TYPE ERROR :
STRUCT
	bError : BOOL;
	nErrorCode : UDINT;
	dtCurrentTime : DT;
END_STRUCT
END_TYPE

(* stored: Version 1.1.0.1
   DUT ERROR: Id {08c499f3-50fc-4f94-95ff-2cf027969d8c} *)
